// TIA Portal V17 export
// export: Created 2024-08-07T21:43:52.9534926Z, ExportSetting WithDefaults, DisplayName Totally Integrated Automation Portal, DisplayVersion V17 Update 7, DisplayName TIA Portal Openness, DisplayVersion V17 Update 7, DisplayName TIA Portal Version Control Interface, DisplayVersion V17, DisplayName SINAMICS Startdrive Advanced, DisplayVersion V17 SP2, DisplayName SINAMICS Startdrive G110M, G120, G120C, G120D, G120P, G115D, DisplayVersion V17 SP2, DisplayName SINAMICS Startdrive G130, G150, S120, S150, SINAMICS MV, S210, DisplayVersion V17 SP2, DisplayName STEP 7 Professional, DisplayVersion V17 Update 7, DisplayName STEP 7 Safety, DisplayVersion V17 Update 6, DisplayName WinCC Advanced / Unified PC, DisplayVersion V17 Update 7
FUNCTION_BLOCK "FB_TurnTable"   // FB3600, LAD
{ S7_Optimized_Access := 'TRUE' }
VERSION : 0.1
// stored: AutoNumber false, IsIECCheckEnabled false, IsRetainMemResEnabled false, MemoryReserve 100, SetENOAutomatically false, UDAEnableTagReadback false
   VAR_INPUT
      iTurnTableInputs : Word;
      iPower : Bool;
      iSafety : Bool;
      iReset : Bool;
      iErrorReset : Bool;
      iManualMode : Bool;
      iAutomaticMode : Bool;
      iTurnTableInSafetyPosition : Bool;
   END_VAR
   VAR_OUTPUT
      qTurnTableOutputs : Word;
      qeCommunication : Bool;
      qeTurnTablePosition : Bool;
      qeTurnTableSafetyPosition : Bool;
      qeTimeout : Bool;
      qePositionRunOver : Bool;
      qeSafety : Bool;
      qeSumError : Bool;
      qeSumWarning : Bool;
   END_VAR
   VAR_IN_OUT
      iqTurnTable : "UDT_TurnTable";
   END_VAR
   VAR
      Edges : Struct
         Enabled : Bool;
         IndexerInPosition : Bool;
      END_STRUCT;
      TONs : Struct
         tDelayCommunication : TON_TIME;
         tDelayPositionError { S7_SetPoint := 'True'} : TON_TIME;
         tDelayErrorReset { S7_SetPoint := 'True'} : TON_TIME;
      END_STRUCT;
   END_VAR
   VAR RETAIN
      RetentiveData : Struct
         LastDirection : Bool;
      END_STRUCT;
   END_VAR
   VAR
      Commands : "UDT_TurnTableCommands";
   END_VAR
   VAR_TEMP
      mode_status : Struct
         manual_mode : Bool;
         automatic_mode : Bool;
         mode_active : Bool;
      END_STRUCT;
      bit : Bool;
      error : Bool;
      ready_to_cw : Bool;
      ready_to_ccw : Bool;
      ready_to_jog : Bool;
      ready_to_start : Bool;
   END_VAR
   VAR_TEMP   // added for the SCL form of the ladder/FBD networks
      _w1 : Bool;
      _w2 : Bool;
      _w3 : Bool;
   END_VAR
BEGIN

REGION Network 1: Read inputs
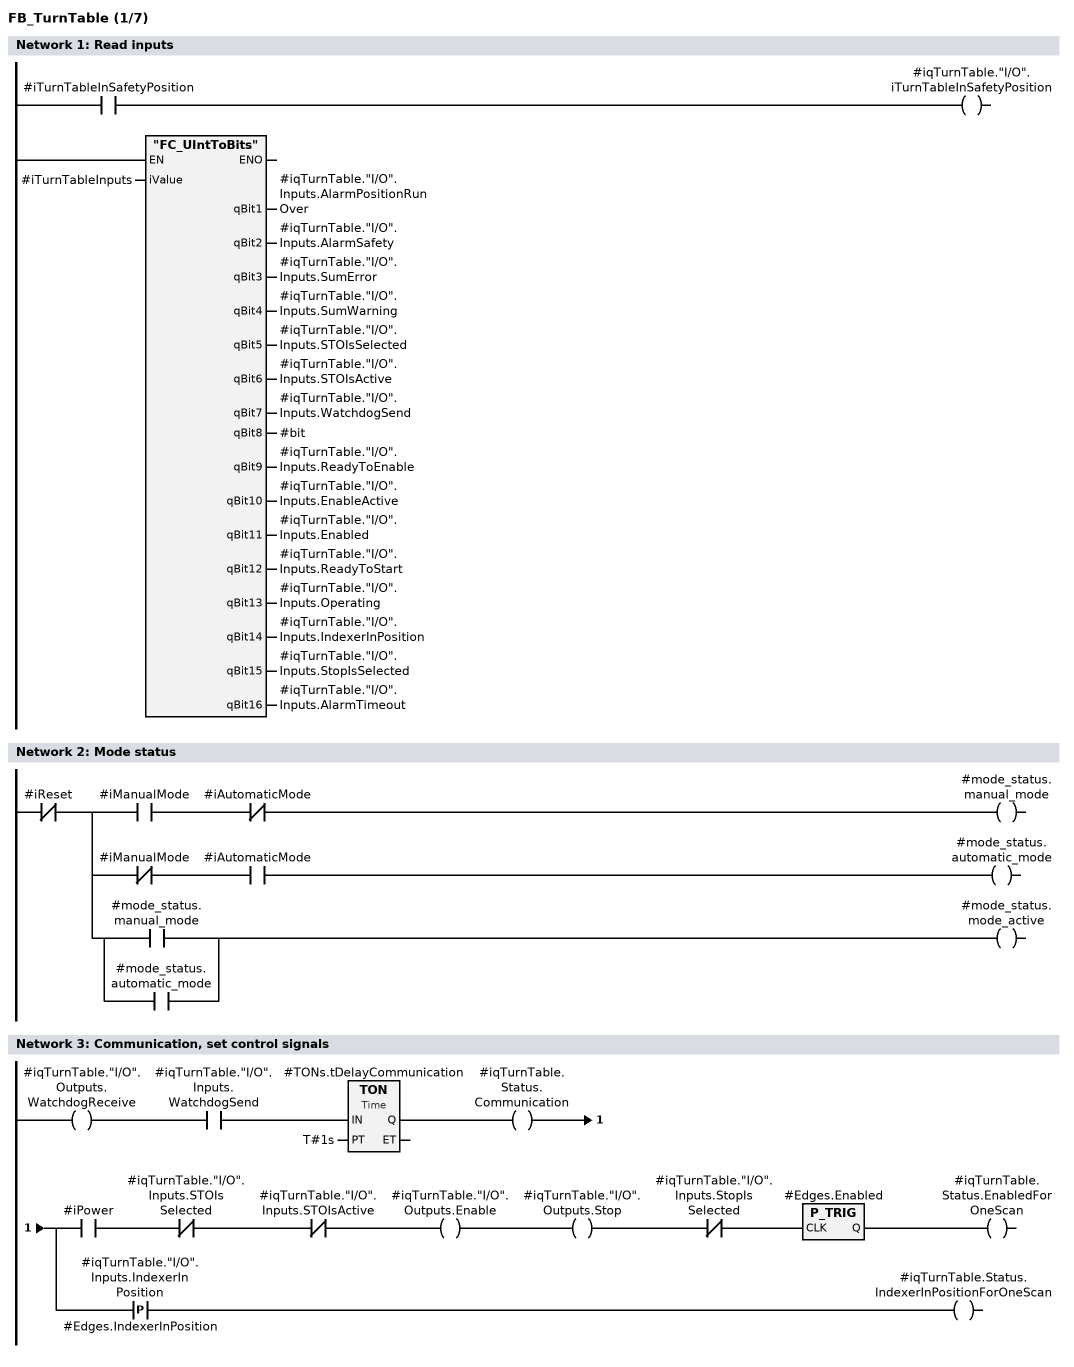
   RUNG wire#powerrail
      Contact( #iTurnTableInSafetyPosition )
      Coil( #iqTurnTable."I/O".iTurnTableInSafetyPosition )
   END_RUNG
   RUNG wire#powerrail
      "FC_UIntToBits"(iValue := #iTurnTableInputs, qBit1 => #iqTurnTable."I/O".Inputs.AlarmPositionRunOver, qBit2 => #iqTurnTable."I/O".Inputs.AlarmSafety, qBit3 => #iqTurnTable."I/O".Inputs.SumError, qBit4 => #iqTurnTable."I/O".Inputs.SumWarning, qBit5 => #iqTurnTable."I/O".Inputs.STOIsSelected, qBit6 => #iqTurnTable."I/O".Inputs.STOIsActive, qBit7 => #iqTurnTable."I/O".Inputs.WatchdogSend, qBit8 => #bit, qBit9 => #iqTurnTable."I/O".Inputs.ReadyToEnable, qBit10 => #iqTurnTable."I/O".Inputs.EnableActive, qBit11 => #iqTurnTable."I/O".Inputs.Enabled, qBit12 => #iqTurnTable."I/O".Inputs.ReadyToStart, qBit13 => #iqTurnTable."I/O".Inputs.Operating, qBit14 => #iqTurnTable."I/O".Inputs.IndexerInPosition, qBit15 => #iqTurnTable."I/O".Inputs.StopIsSelected, qBit16 => #iqTurnTable."I/O".Inputs.AlarmTimeout)
   END_RUNG
   // the same network as SCL:
   #iqTurnTable."I/O".iTurnTableInSafetyPosition := #iTurnTableInSafetyPosition;
   "FC_UIntToBits"(iValue := #iTurnTableInputs,
                   qBit1 => #iqTurnTable."I/O".Inputs.AlarmPositionRunOver,
                   qBit2 => #iqTurnTable."I/O".Inputs.AlarmSafety,
                   qBit3 => #iqTurnTable."I/O".Inputs.SumError,
                   qBit4 => #iqTurnTable."I/O".Inputs.SumWarning,
                   qBit5 => #iqTurnTable."I/O".Inputs.STOIsSelected,
                   qBit6 => #iqTurnTable."I/O".Inputs.STOIsActive,
                   qBit7 => #iqTurnTable."I/O".Inputs.WatchdogSend,
                   qBit8 => #bit,
                   qBit9 => #iqTurnTable."I/O".Inputs.ReadyToEnable,
                   qBit10 => #iqTurnTable."I/O".Inputs.EnableActive,
                   qBit11 => #iqTurnTable."I/O".Inputs.Enabled,
                   qBit12 => #iqTurnTable."I/O".Inputs.ReadyToStart,
                   qBit13 => #iqTurnTable."I/O".Inputs.Operating,
                   qBit14 => #iqTurnTable."I/O".Inputs.IndexerInPosition,
                   qBit15 => #iqTurnTable."I/O".Inputs.StopIsSelected,
                   qBit16 => #iqTurnTable."I/O".Inputs.AlarmTimeout);
END_REGION

REGION Network 2: Mode status
   RUNG wire#powerrail
      I_Contact( #iReset )
      wire#w1
      Contact( #iManualMode )
      I_Contact( #iAutomaticMode )
      Coil( #mode_status.manual_mode )
   END_RUNG
   RUNG wire#w1
      I_Contact( #iManualMode )
      Contact( #iAutomaticMode )
      Coil( #mode_status.automatic_mode )
   END_RUNG
   RUNG wire#w1
      Contact( #mode_status.manual_mode )
      wire#w2
      Coil( #mode_status.mode_active )
   END_RUNG
   RUNG wire#w1
      Contact( #mode_status.automatic_mode )
   END_RUNG wire#w2
   // the same network as SCL:
   #mode_status.manual_mode := NOT #iReset AND #iManualMode AND NOT #iAutomaticMode;
   #mode_status.automatic_mode := NOT #iReset AND NOT #iManualMode AND #iAutomaticMode;
   #mode_status.mode_active := NOT #iReset AND (#mode_status.manual_mode OR #mode_status.automatic_mode);
END_REGION

REGION Network 3: Communication, set control signals
   RUNG wire#powerrail
      Coil( #iqTurnTable."I/O".Outputs.WatchdogReceive )
      Contact( #iqTurnTable."I/O".Inputs.WatchdogSend )
      { S7_Templates := "time_type := Time" } #TONs.tDelayCommunication.TON(pt := T#1s, et =>)
      Coil( #iqTurnTable.Status.Communication )
      wire#w1
      Contact( #iPower )
      I_Contact( #iqTurnTable."I/O".Inputs.STOIsSelected )
      I_Contact( #iqTurnTable."I/O".Inputs.STOIsActive )
      Coil( #iqTurnTable."I/O".Outputs.Enable )
      Coil( #iqTurnTable."I/O".Outputs.Stop )
      I_Contact( #iqTurnTable."I/O".Inputs.StopIsSelected )
      P_Trig( #Edges.Enabled )
      Coil( #iqTurnTable.Status.EnabledForOneScan )
   END_RUNG
   RUNG wire#w1
      P_Contact(operand := #iqTurnTable."I/O".Inputs.IndexerInPosition, bit := #Edges.IndexerInPosition)
      Coil( #iqTurnTable.Status.IndexerInPositionForOneScan )
   END_RUNG
   // the same network as SCL:
   #iqTurnTable."I/O".Outputs.WatchdogReceive := TRUE;
   #TONs.tDelayCommunication.TON(IN := #iqTurnTable."I/O".Inputs.WatchdogSend, PT := T#1s);
   #iqTurnTable.Status.Communication := #TONs.tDelayCommunication.Q;
   #iqTurnTable."I/O".Outputs.Enable := #TONs.tDelayCommunication.Q AND #iPower AND NOT #iqTurnTable."I/O".Inputs.STOIsSelected AND NOT #iqTurnTable."I/O".Inputs.STOIsActive;
   #iqTurnTable."I/O".Outputs.Stop := #iqTurnTable."I/O".Outputs.Enable;
   #_w1 := #iqTurnTable."I/O".Outputs.Enable AND NOT #iqTurnTable."I/O".Inputs.StopIsSelected;
   #_w2 := #_w1 AND NOT #Edges.Enabled;   // rising edge
   #Edges.Enabled := #_w1;
   #iqTurnTable.Status.EnabledForOneScan := #_w2;
   #_w3 := #TONs.tDelayCommunication.Q AND #iqTurnTable."I/O".Inputs.IndexerInPosition AND NOT #Edges.IndexerInPosition;   // rising edge of #iqTurnTable."I/O".Inputs.IndexerInPosition
   #Edges.IndexerInPosition := #iqTurnTable."I/O".Inputs.IndexerInPosition;
   #iqTurnTable.Status.IndexerInPositionForOneScan := #_w3;
END_REGION

REGION Network 4: Errors
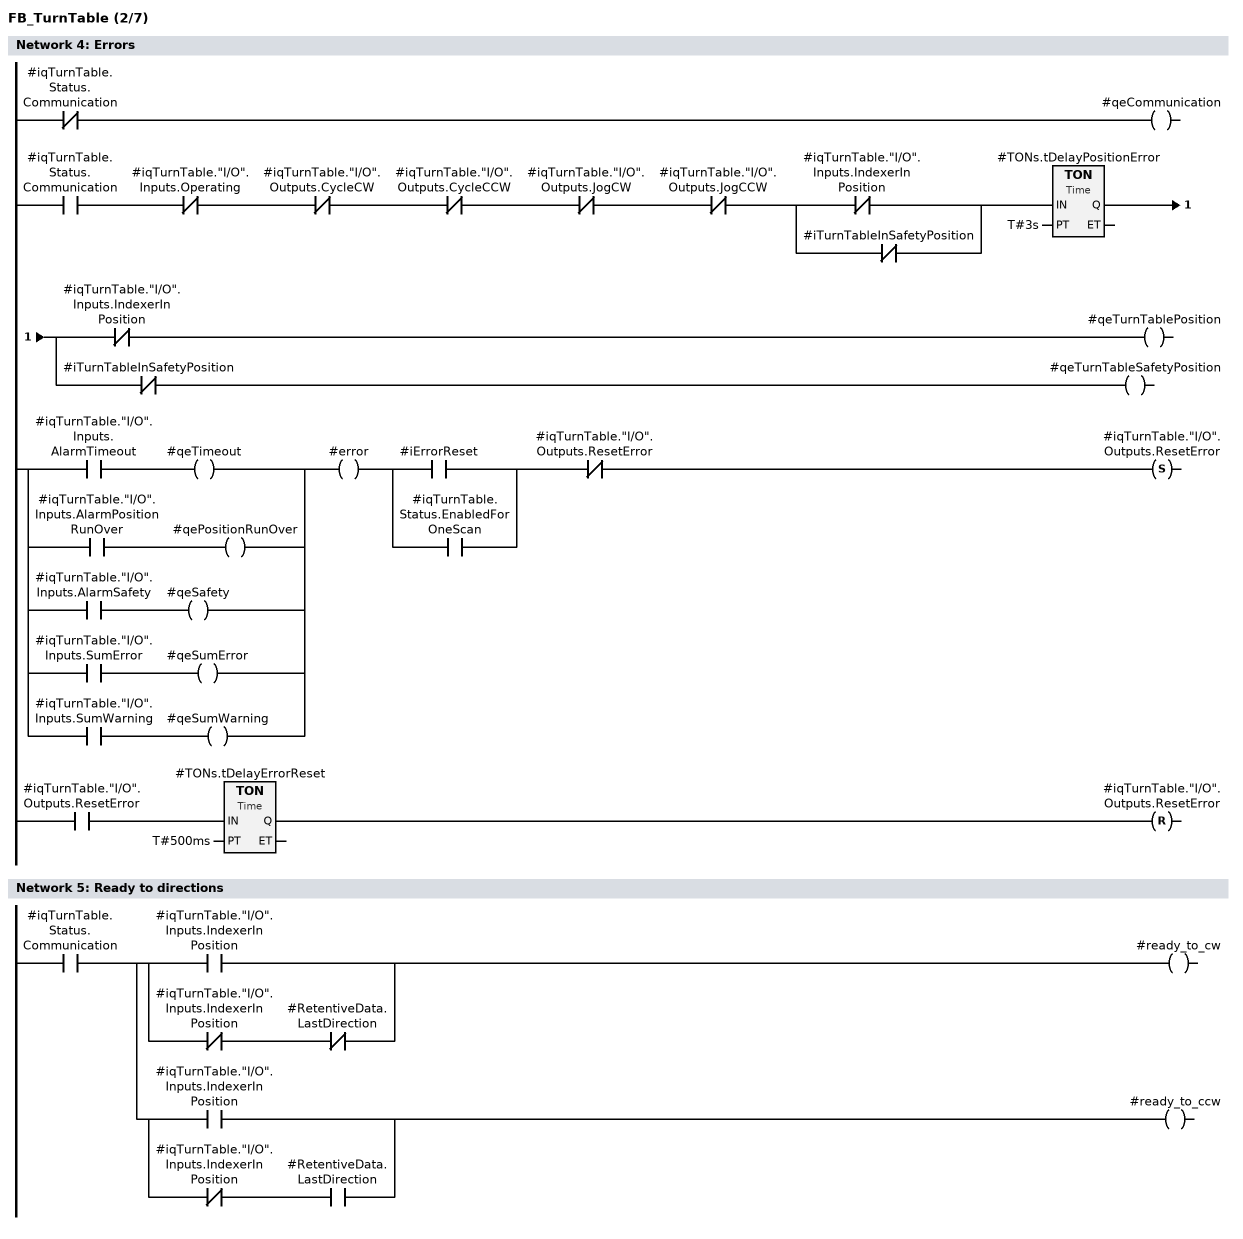
   RUNG wire#powerrail
      I_Contact( #iqTurnTable.Status.Communication )
      Coil( #qeCommunication )
   END_RUNG
   RUNG wire#powerrail
      Contact( #iqTurnTable.Status.Communication )
      I_Contact( #iqTurnTable."I/O".Inputs.Operating )
      I_Contact( #iqTurnTable."I/O".Outputs.CycleCW )
      I_Contact( #iqTurnTable."I/O".Outputs.CycleCCW )
      I_Contact( #iqTurnTable."I/O".Outputs.JogCW )
      I_Contact( #iqTurnTable."I/O".Outputs.JogCCW )
      wire#w1
      I_Contact( #iqTurnTable."I/O".Inputs.IndexerInPosition )
      wire#w2
      { S7_Templates := "time_type := Time" } #TONs.tDelayPositionError.TON(pt := T#3s, et =>)
      wire#w3
      I_Contact( #iqTurnTable."I/O".Inputs.IndexerInPosition )
      Coil( #qeTurnTablePosition )
   END_RUNG
   RUNG wire#w1
      I_Contact( #iTurnTableInSafetyPosition )
   END_RUNG wire#w2
   RUNG wire#w3
      I_Contact( #iTurnTableInSafetyPosition )
      Coil( #qeTurnTableSafetyPosition )
   END_RUNG
   RUNG wire#powerrail
      Contact( #iqTurnTable."I/O".Inputs.AlarmTimeout )
      Coil( #qeTimeout )
      wire#w4
      Coil( #error )
      wire#w5
      Contact( #iErrorReset )
      wire#w6
      I_Contact( #iqTurnTable."I/O".Outputs.ResetError )
      S_Coil( #iqTurnTable."I/O".Outputs.ResetError )
   END_RUNG
   RUNG wire#powerrail
      Contact( #iqTurnTable."I/O".Inputs.AlarmPositionRunOver )
      Coil( #qePositionRunOver )
   END_RUNG wire#w4
   RUNG wire#powerrail
      Contact( #iqTurnTable."I/O".Inputs.AlarmSafety )
      Coil( #qeSafety )
   END_RUNG wire#w4
   RUNG wire#powerrail
      Contact( #iqTurnTable."I/O".Inputs.SumError )
      Coil( #qeSumError )
   END_RUNG wire#w4
   RUNG wire#powerrail
      Contact( #iqTurnTable."I/O".Inputs.SumWarning )
      Coil( #qeSumWarning )
   END_RUNG wire#w4
   RUNG wire#w5
      Contact( #iqTurnTable.Status.EnabledForOneScan )
   END_RUNG wire#w6
   RUNG wire#powerrail
      Contact( #iqTurnTable."I/O".Outputs.ResetError )
      { S7_Templates := "time_type := Time" } #TONs.tDelayErrorReset.TON(pt := T#500ms, et =>)
      R_Coil( #iqTurnTable."I/O".Outputs.ResetError )
   END_RUNG
   // the same network as SCL:
   #qeCommunication := NOT #iqTurnTable.Status.Communication;
   #TONs.tDelayPositionError.TON(IN := #iqTurnTable.Status.Communication AND NOT #iqTurnTable."I/O".Inputs.Operating AND NOT #iqTurnTable."I/O".Outputs.CycleCW AND NOT #iqTurnTable."I/O".Outputs.CycleCCW AND NOT #iqTurnTable."I/O".Outputs.JogCW AND NOT #iqTurnTable."I/O".Outputs.JogCCW AND (NOT #iqTurnTable."I/O".Inputs.IndexerInPosition OR NOT #iTurnTableInSafetyPosition),
                           PT := T#3s);
   #qeTurnTablePosition := #TONs.tDelayPositionError.Q AND NOT #iqTurnTable."I/O".Inputs.IndexerInPosition;
   #qeTurnTableSafetyPosition := #TONs.tDelayPositionError.Q AND NOT #iTurnTableInSafetyPosition;
   #qeTimeout := #iqTurnTable."I/O".Inputs.AlarmTimeout;
   #qePositionRunOver := #iqTurnTable."I/O".Inputs.AlarmPositionRunOver;
   #qeSafety := #iqTurnTable."I/O".Inputs.AlarmSafety;
   #qeSumError := #iqTurnTable."I/O".Inputs.SumError;
   #qeSumWarning := #iqTurnTable."I/O".Inputs.SumWarning;
   #error := #iqTurnTable."I/O".Inputs.AlarmTimeout OR #iqTurnTable."I/O".Inputs.AlarmPositionRunOver OR #iqTurnTable."I/O".Inputs.AlarmSafety OR #iqTurnTable."I/O".Inputs.SumError OR #iqTurnTable."I/O".Inputs.SumWarning;
   IF #error AND (#iErrorReset OR #iqTurnTable.Status.EnabledForOneScan) AND NOT #iqTurnTable."I/O".Outputs.ResetError THEN
       #iqTurnTable."I/O".Outputs.ResetError := TRUE;
   END_IF;
   #TONs.tDelayErrorReset.TON(IN := #iqTurnTable."I/O".Outputs.ResetError, PT := T#500ms);
   IF #TONs.tDelayErrorReset.Q THEN #iqTurnTable."I/O".Outputs.ResetError := FALSE; END_IF;
END_REGION

REGION Network 5: Ready to directions
   RUNG wire#powerrail
      Contact( #iqTurnTable.Status.Communication )
      wire#w1
      Contact( #iqTurnTable."I/O".Inputs.IndexerInPosition )
      wire#w2
      Coil( #ready_to_cw )
   END_RUNG
   RUNG wire#w1
      I_Contact( #iqTurnTable."I/O".Inputs.IndexerInPosition )
      I_Contact( #RetentiveData.LastDirection )
   END_RUNG wire#w2
   RUNG wire#w1
      Contact( #iqTurnTable."I/O".Inputs.IndexerInPosition )
      wire#w3
      Coil( #ready_to_ccw )
   END_RUNG
   RUNG wire#w1
      I_Contact( #iqTurnTable."I/O".Inputs.IndexerInPosition )
      Contact( #RetentiveData.LastDirection )
   END_RUNG wire#w3
   // the same network as SCL:
   #ready_to_cw := #iqTurnTable.Status.Communication AND (#iqTurnTable."I/O".Inputs.IndexerInPosition OR (NOT #iqTurnTable."I/O".Inputs.IndexerInPosition AND NOT #RetentiveData.LastDirection));
   #ready_to_ccw := #iqTurnTable.Status.Communication AND (#iqTurnTable."I/O".Inputs.IndexerInPosition OR (NOT #iqTurnTable."I/O".Inputs.IndexerInPosition AND #RetentiveData.LastDirection));
END_REGION

REGION Network 6: Ready to jog
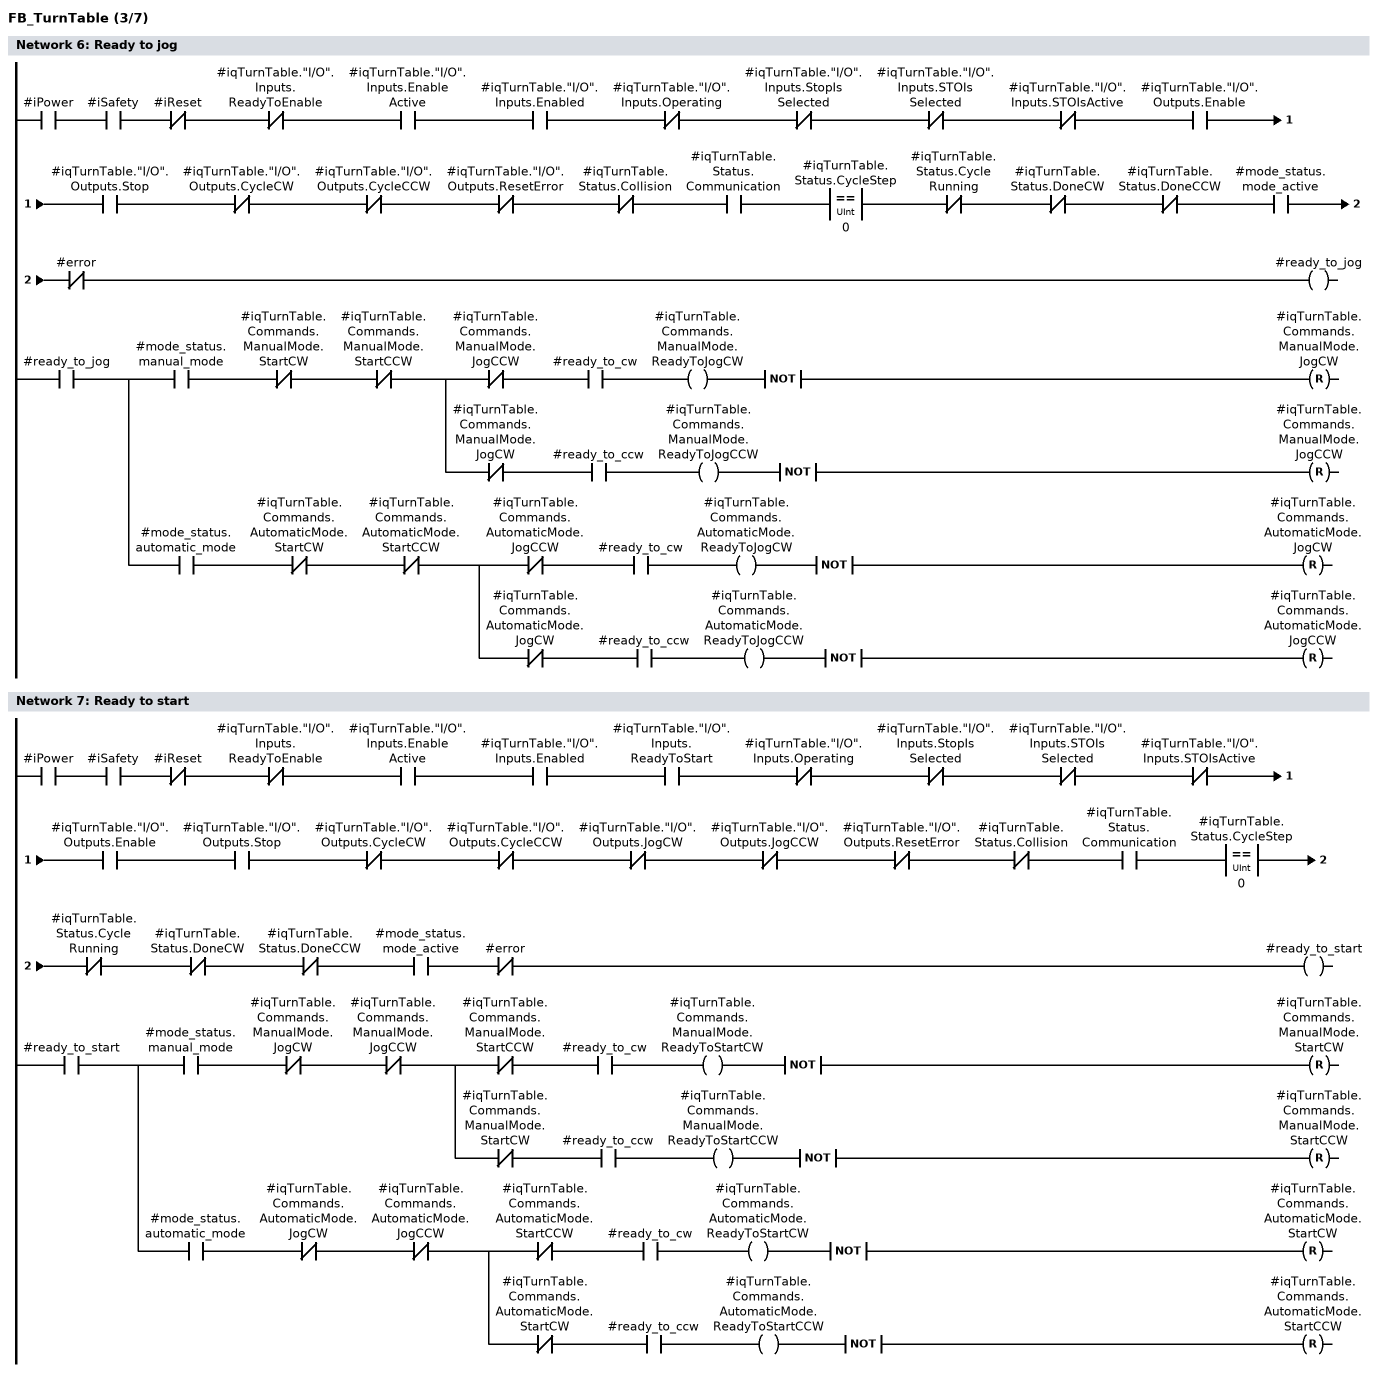
   RUNG wire#powerrail
      Contact( #iPower )
      Contact( #iSafety )
      I_Contact( #iReset )
      I_Contact( #iqTurnTable."I/O".Inputs.ReadyToEnable )
      Contact( #iqTurnTable."I/O".Inputs.EnableActive )
      Contact( #iqTurnTable."I/O".Inputs.Enabled )
      I_Contact( #iqTurnTable."I/O".Inputs.Operating )
      I_Contact( #iqTurnTable."I/O".Inputs.StopIsSelected )
      I_Contact( #iqTurnTable."I/O".Inputs.STOIsSelected )
      I_Contact( #iqTurnTable."I/O".Inputs.STOIsActive )
      Contact( #iqTurnTable."I/O".Outputs.Enable )
      Contact( #iqTurnTable."I/O".Outputs.Stop )
      I_Contact( #iqTurnTable."I/O".Outputs.CycleCW )
      I_Contact( #iqTurnTable."I/O".Outputs.CycleCCW )
      I_Contact( #iqTurnTable."I/O".Outputs.ResetError )
      I_Contact( #iqTurnTable.Status.Collision )
      Contact( #iqTurnTable.Status.Communication )
      { S7_Templates := "SrcType := UInt" } EQ_Contact(in1 := #iqTurnTable.Status.CycleStep, in2 := 0)
      I_Contact( #iqTurnTable.Status.CycleRunning )
      I_Contact( #iqTurnTable.Status.DoneCW )
      I_Contact( #iqTurnTable.Status.DoneCCW )
      Contact( #mode_status.mode_active )
      I_Contact( #error )
      Coil( #ready_to_jog )
   END_RUNG
   RUNG wire#powerrail
      Contact( #ready_to_jog )
      wire#w1
      Contact( #mode_status.manual_mode )
      I_Contact( #iqTurnTable.Commands.ManualMode.StartCW )
      I_Contact( #iqTurnTable.Commands.ManualMode.StartCCW )
      wire#w2
      I_Contact( #iqTurnTable.Commands.ManualMode.JogCCW )
      Contact( #ready_to_cw )
      Coil( #iqTurnTable.Commands.ManualMode.ReadyToJogCW )
      Not()
      R_Coil( #iqTurnTable.Commands.ManualMode.JogCW )
   END_RUNG
   RUNG wire#w2
      I_Contact( #iqTurnTable.Commands.ManualMode.JogCW )
      Contact( #ready_to_ccw )
      Coil( #iqTurnTable.Commands.ManualMode.ReadyToJogCCW )
      Not()
      R_Coil( #iqTurnTable.Commands.ManualMode.JogCCW )
   END_RUNG
   RUNG wire#w1
      Contact( #mode_status.automatic_mode )
      I_Contact( #iqTurnTable.Commands.AutomaticMode.StartCW )
      I_Contact( #iqTurnTable.Commands.AutomaticMode.StartCCW )
      wire#w3
      I_Contact( #iqTurnTable.Commands.AutomaticMode.JogCCW )
      Contact( #ready_to_cw )
      Coil( #iqTurnTable.Commands.AutomaticMode.ReadyToJogCW )
      Not()
      R_Coil( #iqTurnTable.Commands.AutomaticMode.JogCW )
   END_RUNG
   RUNG wire#w3
      I_Contact( #iqTurnTable.Commands.AutomaticMode.JogCW )
      Contact( #ready_to_ccw )
      Coil( #iqTurnTable.Commands.AutomaticMode.ReadyToJogCCW )
      Not()
      R_Coil( #iqTurnTable.Commands.AutomaticMode.JogCCW )
   END_RUNG
   // the same network as SCL:
   #ready_to_jog := #iPower AND #iSafety AND NOT #iReset AND NOT #iqTurnTable."I/O".Inputs.ReadyToEnable AND #iqTurnTable."I/O".Inputs.EnableActive AND #iqTurnTable."I/O".Inputs.Enabled AND NOT #iqTurnTable."I/O".Inputs.Operating AND NOT #iqTurnTable."I/O".Inputs.StopIsSelected AND NOT #iqTurnTable."I/O".Inputs.STOIsSelected AND NOT #iqTurnTable."I/O".Inputs.STOIsActive AND #iqTurnTable."I/O".Outputs.Enable AND #iqTurnTable."I/O".Outputs.Stop AND NOT #iqTurnTable."I/O".Outputs.CycleCW AND NOT #iqTurnTable."I/O".Outputs.CycleCCW AND NOT #iqTurnTable."I/O".Outputs.ResetError AND NOT #iqTurnTable.Status.Collision AND #iqTurnTable.Status.Communication AND (#iqTurnTable.Status.CycleStep = 0) AND NOT #iqTurnTable.Status.CycleRunning AND NOT #iqTurnTable.Status.DoneCW AND NOT #iqTurnTable.Status.DoneCCW AND #mode_status.mode_active AND NOT #error;
   #_w1 := #ready_to_jog AND #mode_status.manual_mode AND NOT #iqTurnTable.Commands.ManualMode.StartCW AND NOT #iqTurnTable.Commands.ManualMode.StartCCW;
   #iqTurnTable.Commands.ManualMode.ReadyToJogCW := #_w1 AND NOT #iqTurnTable.Commands.ManualMode.JogCCW AND #ready_to_cw;
   IF NOT #iqTurnTable.Commands.ManualMode.ReadyToJogCW THEN
       #iqTurnTable.Commands.ManualMode.JogCW := FALSE;
   END_IF;
   #iqTurnTable.Commands.ManualMode.ReadyToJogCCW := #_w1 AND NOT #iqTurnTable.Commands.ManualMode.JogCW AND #ready_to_ccw;
   IF NOT #iqTurnTable.Commands.ManualMode.ReadyToJogCCW THEN
       #iqTurnTable.Commands.ManualMode.JogCCW := FALSE;
   END_IF;
   #_w2 := #ready_to_jog AND #mode_status.automatic_mode AND NOT #iqTurnTable.Commands.AutomaticMode.StartCW AND NOT #iqTurnTable.Commands.AutomaticMode.StartCCW;
   #iqTurnTable.Commands.AutomaticMode.ReadyToJogCW := #_w2 AND NOT #iqTurnTable.Commands.AutomaticMode.JogCCW AND #ready_to_cw;
   IF NOT #iqTurnTable.Commands.AutomaticMode.ReadyToJogCW THEN
       #iqTurnTable.Commands.AutomaticMode.JogCW := FALSE;
   END_IF;
   #iqTurnTable.Commands.AutomaticMode.ReadyToJogCCW := #_w2 AND NOT #iqTurnTable.Commands.AutomaticMode.JogCW AND #ready_to_ccw;
   IF NOT #iqTurnTable.Commands.AutomaticMode.ReadyToJogCCW THEN
       #iqTurnTable.Commands.AutomaticMode.JogCCW := FALSE;
   END_IF;
END_REGION

REGION Network 7: Ready to start
   RUNG wire#powerrail
      Contact( #iPower )
      Contact( #iSafety )
      I_Contact( #iReset )
      I_Contact( #iqTurnTable."I/O".Inputs.ReadyToEnable )
      Contact( #iqTurnTable."I/O".Inputs.EnableActive )
      Contact( #iqTurnTable."I/O".Inputs.Enabled )
      Contact( #iqTurnTable."I/O".Inputs.ReadyToStart )
      I_Contact( #iqTurnTable."I/O".Inputs.Operating )
      I_Contact( #iqTurnTable."I/O".Inputs.StopIsSelected )
      I_Contact( #iqTurnTable."I/O".Inputs.STOIsSelected )
      I_Contact( #iqTurnTable."I/O".Inputs.STOIsActive )
      Contact( #iqTurnTable."I/O".Outputs.Enable )
      Contact( #iqTurnTable."I/O".Outputs.Stop )
      I_Contact( #iqTurnTable."I/O".Outputs.CycleCW )
      I_Contact( #iqTurnTable."I/O".Outputs.CycleCCW )
      I_Contact( #iqTurnTable."I/O".Outputs.JogCW )
      I_Contact( #iqTurnTable."I/O".Outputs.JogCCW )
      I_Contact( #iqTurnTable."I/O".Outputs.ResetError )
      I_Contact( #iqTurnTable.Status.Collision )
      Contact( #iqTurnTable.Status.Communication )
      { S7_Templates := "SrcType := UInt" } EQ_Contact(in1 := #iqTurnTable.Status.CycleStep, in2 := 0)
      I_Contact( #iqTurnTable.Status.CycleRunning )
      I_Contact( #iqTurnTable.Status.DoneCW )
      I_Contact( #iqTurnTable.Status.DoneCCW )
      Contact( #mode_status.mode_active )
      I_Contact( #error )
      Coil( #ready_to_start )
   END_RUNG
   RUNG wire#powerrail
      Contact( #ready_to_start )
      wire#w1
      Contact( #mode_status.manual_mode )
      I_Contact( #iqTurnTable.Commands.ManualMode.JogCW )
      I_Contact( #iqTurnTable.Commands.ManualMode.JogCCW )
      wire#w2
      I_Contact( #iqTurnTable.Commands.ManualMode.StartCCW )
      Contact( #ready_to_cw )
      Coil( #iqTurnTable.Commands.ManualMode.ReadyToStartCW )
      Not()
      R_Coil( #iqTurnTable.Commands.ManualMode.StartCW )
   END_RUNG
   RUNG wire#w2
      I_Contact( #iqTurnTable.Commands.ManualMode.StartCW )
      Contact( #ready_to_ccw )
      Coil( #iqTurnTable.Commands.ManualMode.ReadyToStartCCW )
      Not()
      R_Coil( #iqTurnTable.Commands.ManualMode.StartCCW )
   END_RUNG
   RUNG wire#w1
      Contact( #mode_status.automatic_mode )
      I_Contact( #iqTurnTable.Commands.AutomaticMode.JogCW )
      I_Contact( #iqTurnTable.Commands.AutomaticMode.JogCCW )
      wire#w3
      I_Contact( #iqTurnTable.Commands.AutomaticMode.StartCCW )
      Contact( #ready_to_cw )
      Coil( #iqTurnTable.Commands.AutomaticMode.ReadyToStartCW )
      Not()
      R_Coil( #iqTurnTable.Commands.AutomaticMode.StartCW )
   END_RUNG
   RUNG wire#w3
      I_Contact( #iqTurnTable.Commands.AutomaticMode.StartCW )
      Contact( #ready_to_ccw )
      Coil( #iqTurnTable.Commands.AutomaticMode.ReadyToStartCCW )
      Not()
      R_Coil( #iqTurnTable.Commands.AutomaticMode.StartCCW )
   END_RUNG
   // the same network as SCL:
   #ready_to_start := #iPower AND #iSafety AND NOT #iReset AND NOT #iqTurnTable."I/O".Inputs.ReadyToEnable AND #iqTurnTable."I/O".Inputs.EnableActive AND #iqTurnTable."I/O".Inputs.Enabled AND #iqTurnTable."I/O".Inputs.ReadyToStart AND NOT #iqTurnTable."I/O".Inputs.Operating AND NOT #iqTurnTable."I/O".Inputs.StopIsSelected AND NOT #iqTurnTable."I/O".Inputs.STOIsSelected AND NOT #iqTurnTable."I/O".Inputs.STOIsActive AND #iqTurnTable."I/O".Outputs.Enable AND #iqTurnTable."I/O".Outputs.Stop AND NOT #iqTurnTable."I/O".Outputs.CycleCW AND NOT #iqTurnTable."I/O".Outputs.CycleCCW AND NOT #iqTurnTable."I/O".Outputs.JogCW AND NOT #iqTurnTable."I/O".Outputs.JogCCW AND NOT #iqTurnTable."I/O".Outputs.ResetError AND NOT #iqTurnTable.Status.Collision AND #iqTurnTable.Status.Communication AND (#iqTurnTable.Status.CycleStep = 0) AND NOT #iqTurnTable.Status.CycleRunning AND NOT #iqTurnTable.Status.DoneCW AND NOT #iqTurnTable.Status.DoneCCW AND #mode_status.mode_active AND NOT #error;
   #_w1 := #ready_to_start AND #mode_status.manual_mode AND NOT #iqTurnTable.Commands.ManualMode.JogCW AND NOT #iqTurnTable.Commands.ManualMode.JogCCW;
   #iqTurnTable.Commands.ManualMode.ReadyToStartCW := #_w1 AND NOT #iqTurnTable.Commands.ManualMode.StartCCW AND #ready_to_cw;
   IF NOT #iqTurnTable.Commands.ManualMode.ReadyToStartCW THEN
       #iqTurnTable.Commands.ManualMode.StartCW := FALSE;
   END_IF;
   #iqTurnTable.Commands.ManualMode.ReadyToStartCCW := #_w1 AND NOT #iqTurnTable.Commands.ManualMode.StartCW AND #ready_to_ccw;
   IF NOT #iqTurnTable.Commands.ManualMode.ReadyToStartCCW THEN
       #iqTurnTable.Commands.ManualMode.StartCCW := FALSE;
   END_IF;
   #_w2 := #ready_to_start AND #mode_status.automatic_mode AND NOT #iqTurnTable.Commands.AutomaticMode.JogCW AND NOT #iqTurnTable.Commands.AutomaticMode.JogCCW;
   #iqTurnTable.Commands.AutomaticMode.ReadyToStartCW := #_w2 AND NOT #iqTurnTable.Commands.AutomaticMode.StartCCW AND #ready_to_cw;
   IF NOT #iqTurnTable.Commands.AutomaticMode.ReadyToStartCW THEN
       #iqTurnTable.Commands.AutomaticMode.StartCW := FALSE;
   END_IF;
   #iqTurnTable.Commands.AutomaticMode.ReadyToStartCCW := #_w2 AND NOT #iqTurnTable.Commands.AutomaticMode.StartCW AND #ready_to_ccw;
   IF NOT #iqTurnTable.Commands.AutomaticMode.ReadyToStartCCW THEN
       #iqTurnTable.Commands.AutomaticMode.StartCCW := FALSE;
   END_IF;
END_REGION

REGION Network 8: Set commands
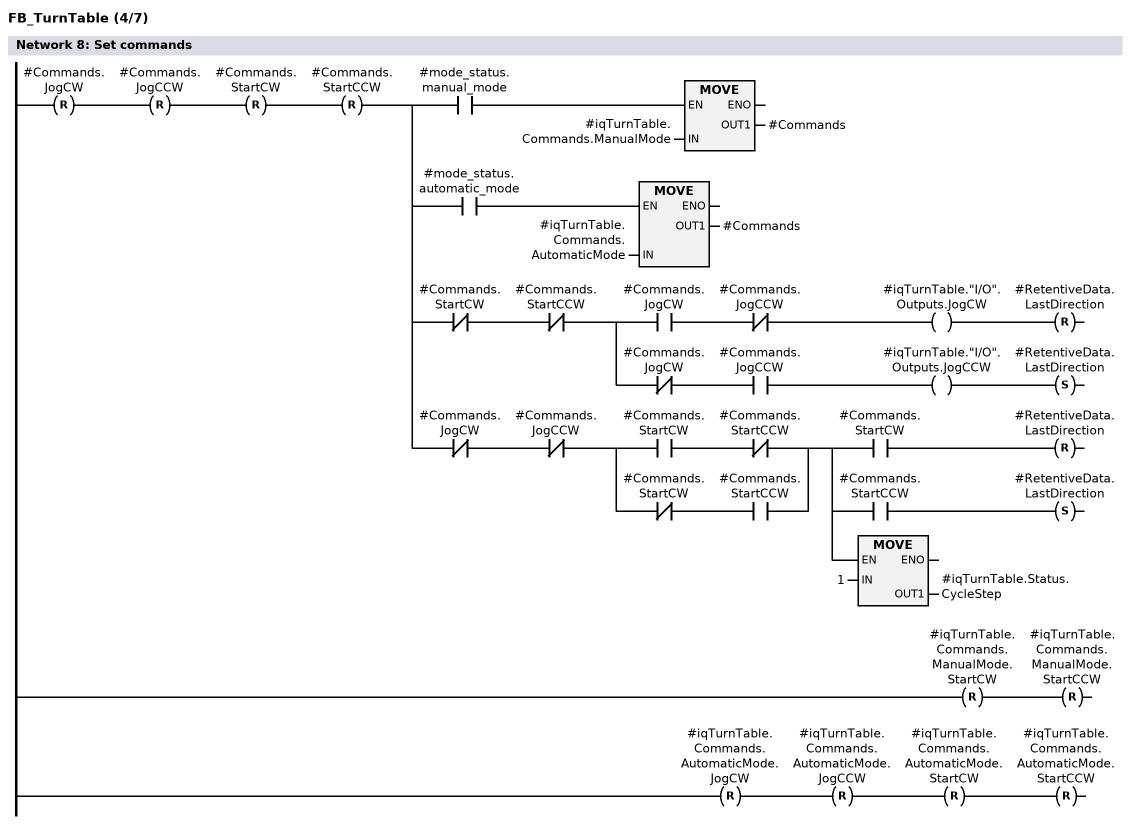
   RUNG wire#powerrail
      R_Coil( #Commands.JogCW )
      R_Coil( #Commands.JogCCW )
      R_Coil( #Commands.StartCW )
      R_Coil( #Commands.StartCCW )
      wire#w1
      Contact( #mode_status.manual_mode )
      Move(in := #iqTurnTable.Commands.ManualMode, out1 => #Commands)
   END_RUNG
   RUNG wire#w1
      Contact( #mode_status.automatic_mode )
      Move(in := #iqTurnTable.Commands.AutomaticMode, out1 => #Commands)
   END_RUNG
   RUNG wire#w1
      I_Contact( #Commands.StartCW )
      I_Contact( #Commands.StartCCW )
      wire#w2
      Contact( #Commands.JogCW )
      I_Contact( #Commands.JogCCW )
      Coil( #iqTurnTable."I/O".Outputs.JogCW )
      R_Coil( #RetentiveData.LastDirection )
   END_RUNG
   RUNG wire#w2
      I_Contact( #Commands.JogCW )
      Contact( #Commands.JogCCW )
      Coil( #iqTurnTable."I/O".Outputs.JogCCW )
      S_Coil( #RetentiveData.LastDirection )
   END_RUNG
   RUNG wire#w1
      I_Contact( #Commands.JogCW )
      I_Contact( #Commands.JogCCW )
      wire#w3
      Contact( #Commands.StartCW )
      I_Contact( #Commands.StartCCW )
      wire#w4
      Contact( #Commands.StartCW )
      R_Coil( #RetentiveData.LastDirection )
   END_RUNG
   RUNG wire#w3
      I_Contact( #Commands.StartCW )
      Contact( #Commands.StartCCW )
   END_RUNG wire#w4
   RUNG wire#w4
      Contact( #Commands.StartCCW )
      S_Coil( #RetentiveData.LastDirection )
   END_RUNG
   RUNG wire#w4
      Move(in := 1, out1 => #iqTurnTable.Status.CycleStep)
   END_RUNG
   RUNG wire#powerrail
      R_Coil( #iqTurnTable.Commands.ManualMode.StartCW )
      R_Coil( #iqTurnTable.Commands.ManualMode.StartCCW )
   END_RUNG
   RUNG wire#powerrail
      R_Coil( #iqTurnTable.Commands.AutomaticMode.JogCW )
      R_Coil( #iqTurnTable.Commands.AutomaticMode.JogCCW )
      R_Coil( #iqTurnTable.Commands.AutomaticMode.StartCW )
      R_Coil( #iqTurnTable.Commands.AutomaticMode.StartCCW )
   END_RUNG
   // the same network as SCL:
   #Commands.JogCW := FALSE;
   #Commands.JogCCW := FALSE;
   #Commands.StartCW := FALSE;
   #Commands.StartCCW := FALSE;
   IF #mode_status.manual_mode THEN #Commands := #iqTurnTable.Commands.ManualMode; END_IF;
   IF #mode_status.automatic_mode THEN #Commands := #iqTurnTable.Commands.AutomaticMode; END_IF;
   #_w1 := NOT #Commands.StartCW AND NOT #Commands.StartCCW;
   #iqTurnTable."I/O".Outputs.JogCW := #_w1 AND #Commands.JogCW AND NOT #Commands.JogCCW;
   IF #iqTurnTable."I/O".Outputs.JogCW THEN #RetentiveData.LastDirection := FALSE; END_IF;
   #iqTurnTable."I/O".Outputs.JogCCW := #_w1 AND NOT #Commands.JogCW AND #Commands.JogCCW;
   IF #iqTurnTable."I/O".Outputs.JogCCW THEN #RetentiveData.LastDirection := TRUE; END_IF;
   #_w2 := NOT #Commands.JogCW AND NOT #Commands.JogCCW AND ((#Commands.StartCW AND NOT #Commands.StartCCW) OR (NOT #Commands.StartCW AND #Commands.StartCCW));
   IF #_w2 AND #Commands.StartCW THEN #RetentiveData.LastDirection := FALSE; END_IF;
   IF #_w2 AND #Commands.StartCCW THEN #RetentiveData.LastDirection := TRUE; END_IF;
   IF #_w2 THEN #iqTurnTable.Status.CycleStep := 1; END_IF;
   #iqTurnTable.Commands.ManualMode.StartCW := FALSE;
   #iqTurnTable.Commands.ManualMode.StartCCW := FALSE;
   #iqTurnTable.Commands.AutomaticMode.JogCW := FALSE;
   #iqTurnTable.Commands.AutomaticMode.JogCCW := FALSE;
   #iqTurnTable.Commands.AutomaticMode.StartCW := FALSE;
   #iqTurnTable.Commands.AutomaticMode.StartCCW := FALSE;
END_REGION

REGION Network 9: Cycle: Reset
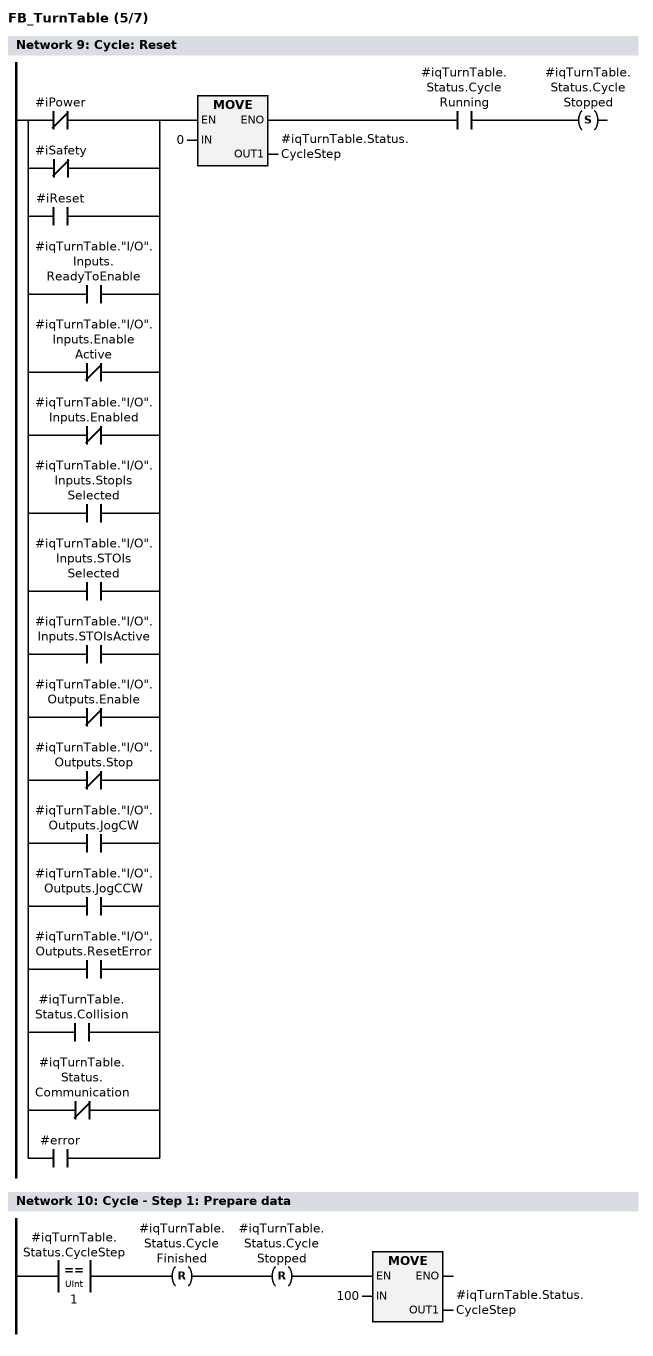
   RUNG wire#powerrail
      I_Contact( #iPower )
      wire#w1
      Move(in := 0, out1 => #iqTurnTable.Status.CycleStep)
      Contact( #iqTurnTable.Status.CycleRunning )
      S_Coil( #iqTurnTable.Status.CycleStopped )
   END_RUNG
   RUNG wire#powerrail
      I_Contact( #iSafety )
   END_RUNG wire#w1
   RUNG wire#powerrail
      Contact( #iReset )
   END_RUNG wire#w1
   RUNG wire#powerrail
      Contact( #iqTurnTable."I/O".Inputs.ReadyToEnable )
   END_RUNG wire#w1
   RUNG wire#powerrail
      I_Contact( #iqTurnTable."I/O".Inputs.EnableActive )
   END_RUNG wire#w1
   RUNG wire#powerrail
      I_Contact( #iqTurnTable."I/O".Inputs.Enabled )
   END_RUNG wire#w1
   RUNG wire#powerrail
      Contact( #iqTurnTable."I/O".Inputs.StopIsSelected )
   END_RUNG wire#w1
   RUNG wire#powerrail
      Contact( #iqTurnTable."I/O".Inputs.STOIsSelected )
   END_RUNG wire#w1
   RUNG wire#powerrail
      Contact( #iqTurnTable."I/O".Inputs.STOIsActive )
   END_RUNG wire#w1
   RUNG wire#powerrail
      I_Contact( #iqTurnTable."I/O".Outputs.Enable )
   END_RUNG wire#w1
   RUNG wire#powerrail
      I_Contact( #iqTurnTable."I/O".Outputs.Stop )
   END_RUNG wire#w1
   RUNG wire#powerrail
      Contact( #iqTurnTable."I/O".Outputs.JogCW )
   END_RUNG wire#w1
   RUNG wire#powerrail
      Contact( #iqTurnTable."I/O".Outputs.JogCCW )
   END_RUNG wire#w1
   RUNG wire#powerrail
      Contact( #iqTurnTable."I/O".Outputs.ResetError )
   END_RUNG wire#w1
   RUNG wire#powerrail
      Contact( #iqTurnTable.Status.Collision )
   END_RUNG wire#w1
   RUNG wire#powerrail
      I_Contact( #iqTurnTable.Status.Communication )
   END_RUNG wire#w1
   RUNG wire#powerrail
      Contact( #error )
   END_RUNG wire#w1
   // the same network as SCL:
   #_w1 := NOT #iPower OR NOT #iSafety OR #iReset OR #iqTurnTable."I/O".Inputs.ReadyToEnable OR NOT #iqTurnTable."I/O".Inputs.EnableActive OR NOT #iqTurnTable."I/O".Inputs.Enabled OR #iqTurnTable."I/O".Inputs.StopIsSelected OR #iqTurnTable."I/O".Inputs.STOIsSelected OR #iqTurnTable."I/O".Inputs.STOIsActive OR NOT #iqTurnTable."I/O".Outputs.Enable OR NOT #iqTurnTable."I/O".Outputs.Stop OR #iqTurnTable."I/O".Outputs.JogCW OR #iqTurnTable."I/O".Outputs.JogCCW OR #iqTurnTable."I/O".Outputs.ResetError OR #iqTurnTable.Status.Collision OR NOT #iqTurnTable.Status.Communication OR #error;
   IF #_w1 THEN #iqTurnTable.Status.CycleStep := 0; END_IF;
   IF #_w1 AND #iqTurnTable.Status.CycleRunning THEN #iqTurnTable.Status.CycleStopped := TRUE; END_IF;
END_REGION

REGION Network 10: Cycle - Step 1: Prepare data
   RUNG wire#powerrail
      { S7_Templates := "SrcType := UInt" } EQ_Contact(in1 := #iqTurnTable.Status.CycleStep, in2 := 1)
      R_Coil( #iqTurnTable.Status.CycleFinished )
      R_Coil( #iqTurnTable.Status.CycleStopped )
      Move(in := 100, out1 => #iqTurnTable.Status.CycleStep)
   END_RUNG
   // the same network as SCL:
   IF #iqTurnTable.Status.CycleStep = 1 THEN
       #iqTurnTable.Status.CycleFinished := FALSE;
       #iqTurnTable.Status.CycleStopped := FALSE;
       #iqTurnTable.Status.CycleStep := 100;
   END_IF;
END_REGION

REGION Network 11: Cycle - Step 100: Check out of position
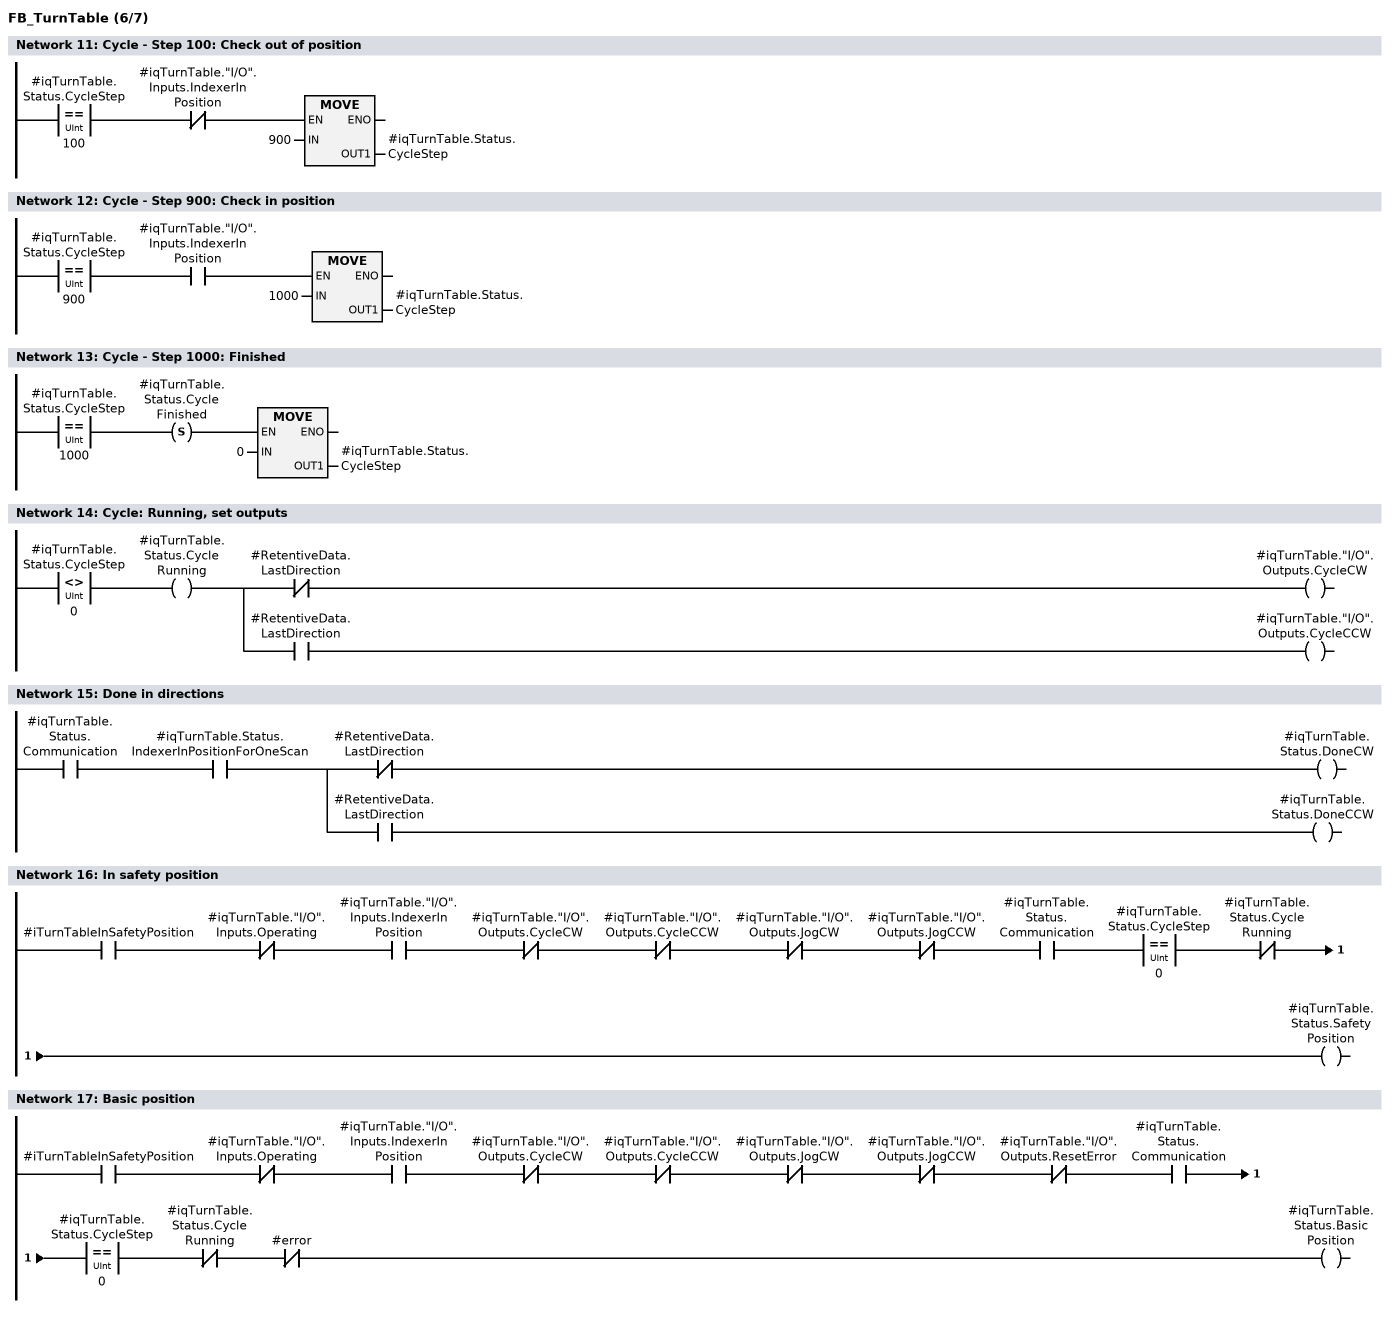
   RUNG wire#powerrail
      { S7_Templates := "SrcType := UInt" } EQ_Contact(in1 := #iqTurnTable.Status.CycleStep, in2 := 100)
      I_Contact( #iqTurnTable."I/O".Inputs.IndexerInPosition )
      Move(in := 900, out1 => #iqTurnTable.Status.CycleStep)
   END_RUNG
   // the same network as SCL:
   IF (#iqTurnTable.Status.CycleStep = 100) AND NOT #iqTurnTable."I/O".Inputs.IndexerInPosition THEN
       #iqTurnTable.Status.CycleStep := 900;
   END_IF;
END_REGION

REGION Network 12: Cycle - Step 900: Check in position
   RUNG wire#powerrail
      { S7_Templates := "SrcType := UInt" } EQ_Contact(in1 := #iqTurnTable.Status.CycleStep, in2 := 900)
      Contact( #iqTurnTable."I/O".Inputs.IndexerInPosition )
      Move(in := 1000, out1 => #iqTurnTable.Status.CycleStep)
   END_RUNG
   // the same network as SCL:
   IF (#iqTurnTable.Status.CycleStep = 900) AND #iqTurnTable."I/O".Inputs.IndexerInPosition THEN
       #iqTurnTable.Status.CycleStep := 1000;
   END_IF;
END_REGION

REGION Network 13: Cycle - Step 1000: Finished
   RUNG wire#powerrail
      { S7_Templates := "SrcType := UInt" } EQ_Contact(in1 := #iqTurnTable.Status.CycleStep, in2 := 1000)
      S_Coil( #iqTurnTable.Status.CycleFinished )
      Move(in := 0, out1 => #iqTurnTable.Status.CycleStep)
   END_RUNG
   // the same network as SCL:
   IF #iqTurnTable.Status.CycleStep = 1000 THEN
       #iqTurnTable.Status.CycleFinished := TRUE;
       #iqTurnTable.Status.CycleStep := 0;
   END_IF;
END_REGION

REGION Network 14: Cycle: Running, set outputs
   RUNG wire#powerrail
      { S7_Templates := "SrcType := UInt" } NE_Contact(in1 := #iqTurnTable.Status.CycleStep, in2 := 0)
      Coil( #iqTurnTable.Status.CycleRunning )
      wire#w1
      I_Contact( #RetentiveData.LastDirection )
      Coil( #iqTurnTable."I/O".Outputs.CycleCW )
   END_RUNG
   RUNG wire#w1
      Contact( #RetentiveData.LastDirection )
      Coil( #iqTurnTable."I/O".Outputs.CycleCCW )
   END_RUNG
   // the same network as SCL:
   #iqTurnTable.Status.CycleRunning := #iqTurnTable.Status.CycleStep <> 0;
   #iqTurnTable."I/O".Outputs.CycleCW := #iqTurnTable.Status.CycleRunning AND NOT #RetentiveData.LastDirection;
   #iqTurnTable."I/O".Outputs.CycleCCW := #iqTurnTable.Status.CycleRunning AND #RetentiveData.LastDirection;
END_REGION

REGION Network 15: Done in directions
   RUNG wire#powerrail
      Contact( #iqTurnTable.Status.Communication )
      Contact( #iqTurnTable.Status.IndexerInPositionForOneScan )
      wire#w1
      I_Contact( #RetentiveData.LastDirection )
      Coil( #iqTurnTable.Status.DoneCW )
   END_RUNG
   RUNG wire#w1
      Contact( #RetentiveData.LastDirection )
      Coil( #iqTurnTable.Status.DoneCCW )
   END_RUNG
   // the same network as SCL:
   #_w1 := #iqTurnTable.Status.Communication AND #iqTurnTable.Status.IndexerInPositionForOneScan;
   #iqTurnTable.Status.DoneCW := #_w1 AND NOT #RetentiveData.LastDirection;
   #iqTurnTable.Status.DoneCCW := #_w1 AND #RetentiveData.LastDirection;
END_REGION

REGION Network 16: In safety position
   RUNG wire#powerrail
      Contact( #iTurnTableInSafetyPosition )
      I_Contact( #iqTurnTable."I/O".Inputs.Operating )
      Contact( #iqTurnTable."I/O".Inputs.IndexerInPosition )
      I_Contact( #iqTurnTable."I/O".Outputs.CycleCW )
      I_Contact( #iqTurnTable."I/O".Outputs.CycleCCW )
      I_Contact( #iqTurnTable."I/O".Outputs.JogCW )
      I_Contact( #iqTurnTable."I/O".Outputs.JogCCW )
      Contact( #iqTurnTable.Status.Communication )
      { S7_Templates := "SrcType := UInt" } EQ_Contact(in1 := #iqTurnTable.Status.CycleStep, in2 := 0)
      I_Contact( #iqTurnTable.Status.CycleRunning )
      Coil( #iqTurnTable.Status.SafetyPosition )
   END_RUNG
   // the same network as SCL:
   #iqTurnTable.Status.SafetyPosition := #iTurnTableInSafetyPosition AND NOT #iqTurnTable."I/O".Inputs.Operating AND #iqTurnTable."I/O".Inputs.IndexerInPosition AND NOT #iqTurnTable."I/O".Outputs.CycleCW AND NOT #iqTurnTable."I/O".Outputs.CycleCCW AND NOT #iqTurnTable."I/O".Outputs.JogCW AND NOT #iqTurnTable."I/O".Outputs.JogCCW AND #iqTurnTable.Status.Communication AND (#iqTurnTable.Status.CycleStep = 0) AND NOT #iqTurnTable.Status.CycleRunning;
END_REGION

REGION Network 17: Basic position
   RUNG wire#powerrail
      Contact( #iTurnTableInSafetyPosition )
      I_Contact( #iqTurnTable."I/O".Inputs.Operating )
      Contact( #iqTurnTable."I/O".Inputs.IndexerInPosition )
      I_Contact( #iqTurnTable."I/O".Outputs.CycleCW )
      I_Contact( #iqTurnTable."I/O".Outputs.CycleCCW )
      I_Contact( #iqTurnTable."I/O".Outputs.JogCW )
      I_Contact( #iqTurnTable."I/O".Outputs.JogCCW )
      I_Contact( #iqTurnTable."I/O".Outputs.ResetError )
      Contact( #iqTurnTable.Status.Communication )
      { S7_Templates := "SrcType := UInt" } EQ_Contact(in1 := #iqTurnTable.Status.CycleStep, in2 := 0)
      I_Contact( #iqTurnTable.Status.CycleRunning )
      I_Contact( #error )
      Coil( #iqTurnTable.Status.BasicPosition )
   END_RUNG
   // the same network as SCL:
   #iqTurnTable.Status.BasicPosition := #iTurnTableInSafetyPosition AND NOT #iqTurnTable."I/O".Inputs.Operating AND #iqTurnTable."I/O".Inputs.IndexerInPosition AND NOT #iqTurnTable."I/O".Outputs.CycleCW AND NOT #iqTurnTable."I/O".Outputs.CycleCCW AND NOT #iqTurnTable."I/O".Outputs.JogCW AND NOT #iqTurnTable."I/O".Outputs.JogCCW AND NOT #iqTurnTable."I/O".Outputs.ResetError AND #iqTurnTable.Status.Communication AND (#iqTurnTable.Status.CycleStep = 0) AND NOT #iqTurnTable.Status.CycleRunning AND NOT #error;
END_REGION

REGION Network 18: Set outputs
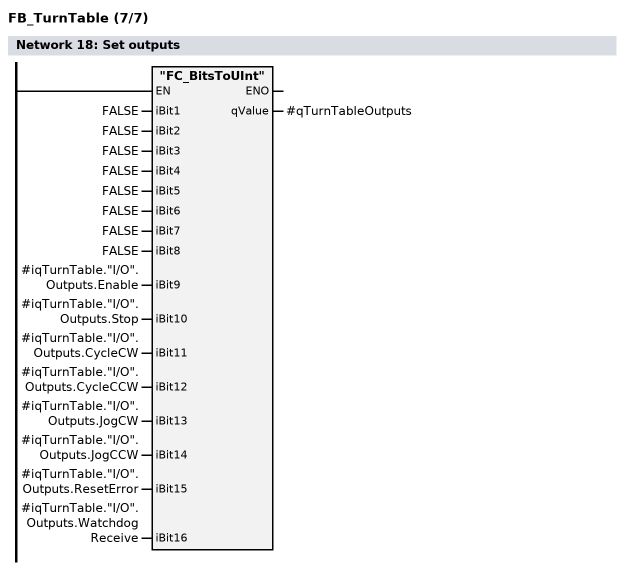
   RUNG wire#powerrail
      "FC_BitsToUInt"(iBit1 := FALSE, iBit2 := FALSE, iBit3 := FALSE, iBit4 := FALSE, iBit5 := FALSE, iBit6 := FALSE, iBit7 := FALSE, iBit8 := FALSE, iBit9 := #iqTurnTable."I/O".Outputs.Enable, iBit10 := #iqTurnTable."I/O".Outputs.Stop, iBit11 := #iqTurnTable."I/O".Outputs.CycleCW, iBit12 := #iqTurnTable."I/O".Outputs.CycleCCW, iBit13 := #iqTurnTable."I/O".Outputs.JogCW, iBit14 := #iqTurnTable."I/O".Outputs.JogCCW, iBit15 := #iqTurnTable."I/O".Outputs.ResetError, iBit16 := #iqTurnTable."I/O".Outputs.WatchdogReceive, qValue => #qTurnTableOutputs)
   END_RUNG
   // the same network as SCL:
   "FC_BitsToUInt"(iBit1 := FALSE,
                   iBit2 := FALSE,
                   iBit3 := FALSE,
                   iBit4 := FALSE,
                   iBit5 := FALSE,
                   iBit6 := FALSE,
                   iBit7 := FALSE,
                   iBit8 := FALSE,
                   iBit9 := #iqTurnTable."I/O".Outputs.Enable,
                   iBit10 := #iqTurnTable."I/O".Outputs.Stop,
                   iBit11 := #iqTurnTable."I/O".Outputs.CycleCW,
                   iBit12 := #iqTurnTable."I/O".Outputs.CycleCCW,
                   iBit13 := #iqTurnTable."I/O".Outputs.JogCW,
                   iBit14 := #iqTurnTable."I/O".Outputs.JogCCW,
                   iBit15 := #iqTurnTable."I/O".Outputs.ResetError,
                   iBit16 := #iqTurnTable."I/O".Outputs.WatchdogReceive,
                   qValue => #qTurnTableOutputs);
END_REGION
END_FUNCTION_BLOCK
